FUNCTION_BLOCK FB_HomeNC_TestDouble IMPLEMENTS I_Home
VAR
	bError : BOOL;
	nErrorID : UDINT := 23000;
END_VAR

{warning 'Add property implementation'}
PROPERTY Aborted : BOOL
GET
END_GET
END_PROPERTY

{warning 'Add property implementation'}
PROPERTY Active : BOOL
GET
END_GET
END_PROPERTY

{warning 'Add property implementation'}
PROPERTY Busy : BOOL
GET
END_GET
END_PROPERTY

{warning 'Add property implementation'}
PROPERTY Done : BOOL
GET
END_GET
END_PROPERTY

{warning 'Add property implementation'}
PROPERTY Error : BOOL
GET
Error := bError;
END_GET
SET
bError := Error;
END_SET
END_PROPERTY

{warning 'Add property implementation'}
PROPERTY ErrorID : UDINT
GET
ErrorId := nErrorID;
END_GET
SET
nErrorId := ErrorID;
END_SET
END_PROPERTY

{warning 'Add property implementation'}
PROPERTY HLDone : BOOL
GET
END_GET
END_PROPERTY

{warning 'Add method implementation '}
METHOD Home
VAR_INPUT
	Position	: LREAL := .DEFAULT_HOME_POSITION;
	BufferMode	: MC_BufferMode;
END_VAR
END_METHOD

{warning 'Add property implementation'}
PROPERTY Message : T_MAXSTRING
GET
END_GET
END_PROPERTY

{warning 'Add property implementation'}
PROPERTY Mode : E_EpicsHomeCmd
GET
END_GET
SET
END_SET
END_PROPERTY

{warning 'Add property implementation'}
PROPERTY Offset : LREAL
SET
END_SET
END_PROPERTY

{warning 'Add property implementation'}
PROPERTY Position : LREAL
SET
END_SET
END_PROPERTY

END_FUNCTION_BLOCK

(* stored: Version 1.1.0.1
   POU FB_HomeNC_TestDouble: Id {92369e88-ac45-4279-8a11-b68694d238eb}, SpecialFunc None
   Property Aborted: Id {c9df4b65-ad0f-4d14-ad65-fb9851ad84d9}
   Get Get: Id {947ca632-6123-4116-a85c-2576822e8f62}
   Property Active: Id {241a6a0e-f9c7-476a-86be-5a72a240a164}
   Get Get: Id {3883dbfa-54e1-410a-a7c9-32896ccd7786}
   Property Busy: Id {9caf7543-ba5d-419f-bb77-15ace6669680}
   Get Get: Id {d0fdd0ca-90b8-40b7-831c-292ed73bd073}
   Property Done: Id {2526c581-55e7-4365-af95-ce96dcc55d1b}
   Get Get: Id {b5c0a3b3-9ab2-4764-a476-f10595dff2e6}
   Property Error: Id {b271a422-5eee-4804-8a92-21ad242e55ec}
   Get Get: Id {61d6217d-c26d-407c-8fa6-1b297afc88a6}
   Set Set: Id {2aacf805-b5c8-4da8-ab3d-c46872bb28d2}
   Property ErrorID: Id {a0eabf90-bd6d-4bc3-8ca6-26c1c71a8324}
   Get Get: Id {ebd1a6ff-0d4b-4e36-94fd-57e95bf3bccc}
   Set Set: Id {cdda61c9-ac19-4f5e-8edd-9d8a3d9f3c1f}
   Property HLDone: Id {5134cf80-87de-4291-9621-7511945c1ddc}
   Get Get: Id {e767267d-6a2c-4f06-96eb-c8d017dad0bd}
   Method Home: Id {bc29fe62-0c4c-48ff-8558-6e754cb5aa62}
   Property Message: Id {d6a17543-0f80-45d3-8181-698680dc3d70}
   Get Get: Id {39d5504e-6ff3-4979-9454-8f507d992ef3}
   Property Mode: Id {477415f6-c414-4767-9416-e8409357d862}
   Get Get: Id {d0c6ac43-f2bf-4458-aef8-1136ed6998ac}
   Set Set: Id {e4189299-a2ff-41b4-9e45-56bd089576ea}
   Property Offset: Id {f41442b8-f272-469b-8426-e8131ed2e6cc}
   Set Set: Id {02f0a801-3026-4ec0-82ac-ce855984faed}
   Property Position: Id {c30c4c65-6691-4080-85b0-79e0e7001911}
   Set Set: Id {0d7dd038-26d9-4b5a-812f-2690a83fcded} *)
